FUNCTION_BLOCK CentralServer (* Basic Function Block Type *)
  (* Standard: 61499-2 *)
  (* Version 0.2, 2003-12-04, JHC, Rockwell Automation, Renamed for better indexing. *)
  (* Version 0.1, 2002-11-05, JHC, Rockwell Automation, Corrected missing ST element in Algorithm REQ. *)
  (* Version 0.0, 2000-05-30, JHC, Rockwell Automation *)
  (* Compiler header: package fb.rt.cs725; *)
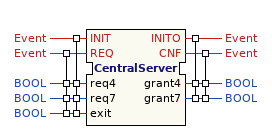
  EVENT_INPUT
    INIT WITH req4, req7, exit; (* Initialization Request *)
    REQ WITH req4, req7, exit; (* Normal Execution Request *)
  END_EVENT
  EVENT_OUTPUT
    INITO WITH grant4, grant7; (* Initialization Confirm *)
    CNF WITH grant7, grant4; (* Execution Confirmation *)
  END_EVENT
  VAR_INPUT
    req4 : BOOL; (* Input event qualifier *)
    req7 : BOOL;
    exit : BOOL;
  END_VAR
  VAR_OUTPUT
    grant4 : BOOL;
    grant7 : BOOL;
  END_VAR
  VAR
    firstReq : INT := 0;
    secReq : INT := 0;
    bagInCs : BOOL := false;
  END_VAR
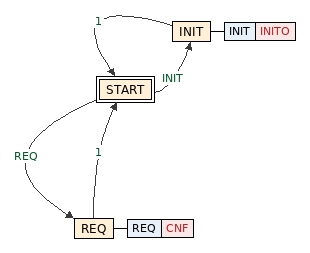
  EC_STATES
    START; (* Initial State *)
    INIT : INIT -> INITO; (* Initialization *)
    REQ : REQ -> CNF; (* Normal execution *)
  END_STATES
  EC_TRANSITIONS
    START TO INIT := INIT;
    INIT TO START := 1;
    REQ TO START := 1;
    START TO REQ := REQ;
  END_TRANSITIONS
  ALGORITHM INIT IN Java: (* Initialization algorithm *)
grant4.value=false;
grant7.value=false;
  END_ALGORITHM
  ALGORITHM REQ IN Java: (* Normally executed algorithm *)
if (!exit.value) {
    bagInCS.value = false;
}
if (req4.value) {
    if (firstReq.value == 0) {
        firstReq.value = 4;
    }
    else {
        secReq.value = 4;
    }
}
if (req7.value) {
    if (firstReq.value == 0) {
        firstReq.value = 7;
    }
    else {
        secReq.value = 7;
    }
}
if (!bagInCs.value) {
    if (firstReq.value == 4) {
        grant4.value = true;
        grant7.value = false;
        firstReq.value = secReq.value;
    }
    else if (firstReq.value == 7) {
        grant4.value = false;
        grant7.value = true;
        firstReq.value = secReq.value;
    }
    else {
        grant4.value = false;
        grant7.value = false;
    }
}
  END_ALGORITHM
END_FUNCTION_BLOCK
